{attribute 'GeneratedUsingTerminal: EL5032-0000-0021'}
{attribute addProperty BoxType "EL5032-0000-0021"}
{attribute addProperty Id "StatusAT %I*Status_81FEA7676PositionAT %I*ULINT8"}
{attribute addProperty CRC "1946487176"}
{attribute addProperty Size "14"}
TYPE FB_Inputs_Channel_74050988 EXTENDS InputBase_8311D824 :
STRUCT
	{attribute addProperty Name "Status"}
	Status AT %I* : Status_81FEA767;
	{attribute addProperty Name "Position"}
	Position AT %I* : ULINT;
END_STRUCT
END_TYPE

(* stored: Version 1.2.0.0, ProductVersion 3.1.4024.9
   DUT FB_Inputs_Channel_74050988: Id {773d01b3-2b33-4f02-95a4-38238967e068} *)
